(* IEC 61131-3 sources: programs/VI-54/VI-54_20171205/VI-54_20171205/Stations/Screen/LseClass170718/Class/FolderDefine, 1 file *)

(* ---- FolderDefine.st ---- *)
(*!
<Class
	Name               = "FolderDefine"
	Revision           = "1.0"
	RealtimeTask       = "false"
	CyclicTask         = "false"
	BackgroundTask     = "false"
	Sigmatek           = "false"
	OSInterface        = "false"
	HighPriority       = "false"
	Automatic          = "false"
	UpdateMode         = "Prescan"
	SharedCommandTable = "true"
	Objectsize         = "(690,180)"
	Comment            = "Use this class to add a folder for the diagnostic export.">
	<Channels>
		<Server Name="ClassSvr" Visualized="false" Initialize="false" WriteProtected="true" Retentive="false"/>
		<Server Name="sUserDPNE" Class="StringInternal" Visualized="false" Initialize="true" WriteProtected="false" Retentive="false" Comment="Name + path of the folder. (for example: &quot;C:\MyFolder&quot;)"/>
		<Client Name="cFFHandler" Required="true" Internal="false" Comment="This client has to be connected to an object of the class DiagnosticStationFileFolderHandler."/>
		<Client Name="UserDPNE" Required="true" Internal="true"/>
	</Channels>
	<RevDoku>
		<Owner Company="Sigmatek"/>
		<Dokumentation Revision="1.0" Date="2016-04-25" Author="GreJoh" Company="Sigmatek" Description="Creation"/>
	</RevDoku>
	<Network Name="FolderDefine">
		<!-- List of Components in this network -->
		<Components>
			<Object
				Name       = "UserDPNE"
				Class      = "String"
				Position   = "(120,240)"
				Visualized = "true"
				Remotely   = "true">
				<Channels>
					<Server Name="Data"/>
					<Client Name="SingleRealloc" Value="1"/>
				</Channels>
			</Object>
		</Components>
		<Comments>
		</Comments>
		<!-- List of Connections in this network -->
		<Connections>
			<Connection Source="this.UserDPNE" Destination="UserDPNE.Data"/>
			<Connection Source="this.sUserDPNE" Destination="UserDPNE.Data" Vertices="(848,270),(676,330),"/>
		</Connections>
		<!-- Headerfiles -->
		<Options>
		</Options>
	</Network>
</Class>
*)
FolderDefine : CLASS
  //Servers:
	ClassSvr 	: SvrChCmd_DINT;
	sUserDPNE 	: SvrChCmd_UDINT;
  //Clients:
	UserDPNE 	: CltChCmd_String;
	cFFHandler 	: CltChCmd_DiagnosticStationFileFolderHandler;
  //Variables:
  //Functions:

	FUNCTION VIRTUAL GLOBAL Init;
  //Tables:
	FUNCTION @STD
		VAR_OUTPUT
			ret_code	: CONFSTATES;
		END_VAR;
	FUNCTION GLOBAL TAB @CT_;
END_CLASS;

#pragma using String
#pragma usingLtd DiagnosticStationFileFolderHandler

FUNCTION VIRTUAL GLOBAL FolderDefine::Init
  VAR
    tmpLength : udint;
    tmpDPNE : array [0..199] of char;
  END_VAR

  if _FirstScan then
    tmpLength := UserDPNE.GetLength();
    UserDPNE.ReadDataOff(udOff:=0, pData:=#tmpDPNE[0], udMax:= sizeof(tmpDPNE));
    tmpDPNE[tmpLength] :=0;
    cFFHandler.AddFileFolder(pDPNE:=#tmpDPNE[0], IsFile:=FALSE);
  end_if;

END_FUNCTION
